// TIA Portal V20 export
FUNCTION_BLOCK "FB_Parameters"   // FB64, SCL
{ S7_Optimized_Access := 'TRUE' }
// stored: MemoryReserve 100, SetENOAutomatically false
   VAR
      Shuttle1Enable : "UDT_BoolEnable";
      Shuttle2Enable : Bool;
   END_VAR
   VAR RETAIN
      GazPressureManual : Real := 0.7;   // @Precision:3 @Unit:bar @Min:0.5 @Max:1.2
   END_VAR
   VAR
      CoolingVentilatorSetpoint : Real;
      TemperatureCoolingSetpoint : Real;
      BlowingSetpoint : Real;
      sPresenceShuttle1UndrilledPart : "FB_HMI_PLC_Pos";
      sPresenceShuttle1UndrilledBw { S7_SetPoint := 'True'} : "FB_HMI_PLC_Pos";
      sPresenceShuttle1DrilledPart { S7_SetPoint := 'True'} : "FB_HMI_PLC_Pos";
      sPresenceShuttle1DrilledBw { S7_SetPoint := 'True'} : "FB_HMI_PLC_Pos";
      sPresenceShuttle2UndrilledPart : "FB_HMI_PLC_Pos";
      sPresenceShuttle2UndrilledBw { S7_SetPoint := 'True'} : "FB_HMI_PLC_Pos";
      sPresenceShuttle2DrilledPart { S7_SetPoint := 'True'} : "FB_HMI_PLC_Pos";
      sPresenceShuttle2DrilledBw { S7_SetPoint := 'True'} : "FB_HMI_PLC_Pos";
      sPresenceGripperUndrilledPart : "FB_HMI_PLC_Pos";
      sPresenceGripperUndrilledBw { S7_SetPoint := 'True'} : "FB_HMI_PLC_Pos";
      sPresenceGripperDrilledPart { S7_SetPoint := 'True'} : "FB_HMI_PLC_Pos";
      sPresenceGripperDrilledBw { S7_SetPoint := 'True'} : "FB_HMI_PLC_Pos";
      sPresenceFixtureUndrilledPart : "FB_HMI_PLC_Pos";
      sPresenceFixtureUndrilledBw { S7_SetPoint := 'True'} : "FB_HMI_PLC_Pos";
      sPresenceFixtureDrilledPart { S7_SetPoint := 'True'} : "FB_HMI_PLC_Pos";
      sPresenceFixtureDrilledBw { S7_SetPoint := 'True'} : "FB_HMI_PLC_Pos";
      sHmiChangeEnable { S7_SetPoint := 'True'} : Bool;
   END_VAR
BEGIN
   REGION Description header 
       //==================================================================================
       // POSALUX Swiss SA / (C) Copyright 2025
       //----------------------------------------------------------------------------------
       // Title: FB_OPC_Parameters
       // Comment/Function: 
       // Author: Fabien WALDT
       // Engineering: TIA Portal v20
       //----------------------------------------------------------------------------------
       // Change log table:
       // Version  | Date     | Expert in charge | Changes applied
       // ---------|----------|------------------|-----------------------------------------
       // 00.00.01 | 20260304 | WFA              | First released version
       // =================================================================================
   END_REGION

   REGION Set Points (HMI -> PLC)
       "DB_HMISetting".GasAssistSetPoint := "DB_OPC_Machine".Parameters.GasAssistSetPoint;
       "DB_HMISetting".CoolingVentilatorSetpoint := "DB_OPC_Machine".Parameters.CoolingVentilatorSetpoint;
       "DB_HMISetting".TemperatureCoolingSetpoint := "DB_OPC_Machine".Parameters.TemperatureCoolingSetpoint;
       "DB_HMISetting".BlowingSetpoint := "DB_OPC_Machine".Parameters.BlowingSetpoint;
   END_REGION

   REGION Shuttle Enable (HMI -> PLC)
       "DB_OPC_Machine".Parameters.Shuttle1Enable.IsEnabled := NOT "DB_LoaderShuttle1".sMain.iJobReq AND NOT "DB_LoaderShuttle2".sMain.iJobReq;
       "DB_OPC_Machine".Parameters.Shuttle2Enable.IsEnabled := NOT "DB_LoaderShuttle1".sMain.iJobReq AND NOT "DB_LoaderShuttle2".sMain.iJobReq;

       "DB_HMISetting".Shuttle1Enable := "DB_OPC_Machine".Parameters.Shuttle1Enable.Value;
       "DB_HMISetting".Shuttle2Enable := "DB_OPC_Machine".Parameters.Shuttle2Enable.Value;
   END_REGION

   REGION Sequence
       // Shuttle 1
       "DB_OPC_Machine".Parameters.Sequence.Shuttle1.Main := "DB_LoaderShuttle1".sMain.sCurrent_Step_NB;
       "DB_OPC_Machine".Parameters.Sequence.Shuttle1.ShuttleInt := "DB_LoaderShuttle1".sShuttleInt.sCurrent_Step_NB;
       "DB_OPC_Machine".Parameters.Sequence.Shuttle1.ShuttleExt := "DB_LoaderShuttle1".sShuttleExt.sCurrent_Step_NB;
       "DB_OPC_Machine".Parameters.Sequence.Shuttle1.ControlIn := "DB_LoaderShuttle1".sControlIn.sCurrent_Step_NB;
       "DB_OPC_Machine".Parameters.Sequence.Shuttle1.ControlOut := "DB_LoaderShuttle1".sControlOut.sCurrent_Step_NB;
       "DB_OPC_Machine".Parameters.Sequence.Shuttle1.Blowing := "DB_LoaderShuttle1".sBlowing.sCurrent_Step_NB;
       "DB_OPC_Machine".Parameters.Sequence.Shuttle1.IntLoadUnload := "DB_LoaderShuttle1".sIntLoadUnload.sCurrent_Step_NB;
       "DB_OPC_Machine".Parameters.Sequence.Shuttle1.ExtLoadUnload := "DB_LoaderShuttle1".sExtLoadUnload.sCurrent_Step_NB;
       "DB_OPC_Machine".Parameters.Sequence.Shuttle1.BwLoadUnload := "DB_LoaderShuttle1".sBwLoadUnload.sCurrent_Step_NB;
       "DB_OPC_Machine".Parameters.Sequence.Shuttle1.BwControlIn := "DB_LoaderShuttle1".sBwControlIn.sCurrent_Step_NB;
       "DB_OPC_Machine".Parameters.Sequence.Shuttle1.ActControlIn := "DB_LoaderShuttle1".sActPartControlIn.sCurrent_Step_NB;
       "DB_OPC_Machine".Parameters.Sequence.Shuttle1.ActControlOut := "DB_LoaderShuttle1".sActPartControlOut.sCurrent_Step_NB;
       "DB_OPC_Machine".Parameters.Sequence.Shuttle1.ActBwControlIn := "DB_LoaderShuttle1".sActBwControlIn.sCurrent_Step_NB;

       // Shuttle 2
       "DB_OPC_Machine".Parameters.Sequence.Shuttle2.Main := "DB_LoaderShuttle2".sMain.sCurrent_Step_NB;
       "DB_OPC_Machine".Parameters.Sequence.Shuttle2.ShuttleInt := "DB_LoaderShuttle2".sShuttleInt.sCurrent_Step_NB;
       "DB_OPC_Machine".Parameters.Sequence.Shuttle2.ShuttleExt := "DB_LoaderShuttle2".sShuttleExt.sCurrent_Step_NB;
       "DB_OPC_Machine".Parameters.Sequence.Shuttle2.ControlIn := "DB_LoaderShuttle2".sControlIn.sCurrent_Step_NB;
       "DB_OPC_Machine".Parameters.Sequence.Shuttle2.ControlOut := "DB_LoaderShuttle2".sControlOut.sCurrent_Step_NB;
       "DB_OPC_Machine".Parameters.Sequence.Shuttle2.Blowing := "DB_LoaderShuttle2".sBlowing.sCurrent_Step_NB;
       "DB_OPC_Machine".Parameters.Sequence.Shuttle2.IntLoadUnload := "DB_LoaderShuttle2".sIntLoadUnload.sCurrent_Step_NB;
       "DB_OPC_Machine".Parameters.Sequence.Shuttle2.ExtLoadUnload := "DB_LoaderShuttle2".sExtLoadUnload.sCurrent_Step_NB;
       "DB_OPC_Machine".Parameters.Sequence.Shuttle2.BwLoadUnload := "DB_LoaderShuttle2".sBwLoadUnload.sCurrent_Step_NB;
       "DB_OPC_Machine".Parameters.Sequence.Shuttle2.BwControlIn := "DB_LoaderShuttle2".sBwControlIn.sCurrent_Step_NB;
       "DB_OPC_Machine".Parameters.Sequence.Shuttle2.ActControlIn := "DB_LoaderShuttle2".sActPartControlIn.sCurrent_Step_NB;
       "DB_OPC_Machine".Parameters.Sequence.Shuttle2.ActControlOut := "DB_LoaderShuttle2".sActPartControlout.sCurrent_Step_NB;
       "DB_OPC_Machine".Parameters.Sequence.Shuttle2.ActBwControlIn := "DB_LoaderShuttle2".sActBwControlIn.sCurrent_Step_NB;

       // Fixture
       "DB_OPC_Machine".Parameters.Sequence.Fixture.Blowing := "DB_LoaderFixture".sFixtureBlowing.sCurrent_Step_NB;
       "DB_OPC_Machine".Parameters.Sequence.Fixture.Loading := "DB_LoaderFixture".sFixtureLoading.sCurrent_Step_NB;
       "DB_OPC_Machine".Parameters.Sequence.Fixture.Unloading := "DB_LoaderFixture".sFixtureUnloading.sCurrent_Step_NB;
       "DB_OPC_Machine".Parameters.Sequence.Fixture.V_Init := "DB_LoaderFixture".sFixtureV_Init.sCurrent_Step_NB;
       "DB_OPC_Machine".Parameters.Sequence.Fixture.W_Init := "DB_LoaderFixture".sFixtureW_Init.sCurrent_Step_NB;

   END_REGION

   REGION Presence
       // Shuttle 1
        "DB_OPC_Machine".Parameters.Presence.Shuttle1UndrilledPart := "DB_PartManagement".sPosition.sShuttle1.Undrilled.Presence.Part;
        "DB_OPC_Machine".Parameters.Presence.Shuttle1UndrilledBw := "DB_PartManagement".sPosition.sShuttle1.Undrilled.Presence.BW;
        "DB_OPC_Machine".Parameters.Presence.Shuttle1DrilledPart := "DB_PartManagement".sPosition.sShuttle1.Drilled.Presence.Part;
        "DB_OPC_Machine".Parameters.Presence.Shuttle1DrilledBw := "DB_PartManagement".sPosition.sShuttle1.Drilled.Presence.BW;

       // Shuttle 2
       "DB_OPC_Machine".Parameters.Presence.Shuttle2UndrilledPart := "DB_PartManagement".sPosition.sShuttle2.Undrilled.Presence.Part;
       "DB_OPC_Machine".Parameters.Presence.Shuttle2UndrilledBw := "DB_PartManagement".sPosition.sShuttle2.Undrilled.Presence.BW;
       "DB_OPC_Machine".Parameters.Presence.Shuttle2DrilledPart := "DB_PartManagement".sPosition.sShuttle2.Drilled.Presence.Part;
       "DB_OPC_Machine".Parameters.Presence.Shuttle2DrilledBw := "DB_PartManagement".sPosition.sShuttle2.Drilled.Presence.BW;

       // Gripper
       "DB_OPC_Machine".Parameters.Presence.GripperUndrilledPart := "DB_PartManagement".sPosition.sGripper.Undrilled.Presence.Part;
       "DB_OPC_Machine".Parameters.Presence.GripperUndrilledBw := "DB_PartManagement".sPosition.sGripper.Undrilled.Presence.BW;
       "DB_OPC_Machine".Parameters.Presence.GripperDrilledPart := "DB_PartManagement".sPosition.sGripper.Drilled.Presence.Part;
       "DB_OPC_Machine".Parameters.Presence.GripperDrilledBw := "DB_PartManagement".sPosition.sGripper.Drilled.Presence.BW;

       // Fixture
       "DB_OPC_Machine".Parameters.Presence.FixtureUndrilledPart := "DB_PartManagement".sPosition.sFixture.Undrilled.Presence.Part;
       "DB_OPC_Machine".Parameters.Presence.FixtureUndrilledBw := "DB_PartManagement".sPosition.sFixture.Undrilled.Presence.BW;
       "DB_OPC_Machine".Parameters.Presence.FixtureDrilledPart := "DB_PartManagement".sPosition.sFixture.Drilled.Presence.Part;
       "DB_OPC_Machine".Parameters.Presence.FixtureDrilledBw := "DB_PartManagement".sPosition.sFixture.Drilled.Presence.BW;
   END_REGION

   REGION Presence V2
       // // Shuttle 1
       // #sPresenceShuttle1UndrilledPart("HMI_Change Enable" := #sHmiChangeEnable,
       //                                 ioPLC_State := "DB_PartManagement".sPosition.sShuttle1.Undrilled.Presence.Part,
       //                                 ioHMI_State := "DB_OPC_Machine".Parameters.Presence.Shuttle1UndrilledPart);

       // #sPresenceShuttle1UndrilledBw("HMI_Change Enable" := #sHmiChangeEnable,
       //                               ioPLC_State := "DB_PartManagement".sPosition.sShuttle1.Undrilled.Presence.BW,
       //                               ioHMI_State := "DB_OPC_Machine".Parameters.Presence.Shuttle1UndrilledBw);

       // #sPresenceShuttle1DrilledPart("HMI_Change Enable" := #sHmiChangeEnable,
       //                                 ioPLC_State := "DB_PartManagement".sPosition.sShuttle1.Drilled.Presence.Part,
       //                                 ioHMI_State := "DB_OPC_Machine".Parameters.Presence.Shuttle1DrilledPart);

       // #sPresenceShuttle1DrilledBw("HMI_Change Enable" := #sHmiChangeEnable,
       //                               ioPLC_State := "DB_PartManagement".sPosition.sShuttle1.Drilled.Presence.BW,
       //                               ioHMI_State := "DB_OPC_Machine".Parameters.Presence.Shuttle1DrilledBw);

       //  // Shuttle 2
       //  #sPresenceShuttle2UndrilledPart("HMI_Change Enable" := #sHmiChangeEnable,
       //                                  ioPLC_State := "DB_PartManagement".sPosition.sShuttle2.Undrilled.Presence.Part,
       //                                  ioHMI_State := "DB_OPC_Machine".Parameters.Presence.Shuttle2UndrilledPart);

       //  #sPresenceShuttle2UndrilledBw("HMI_Change Enable" := #sHmiChangeEnable,
       //                                ioPLC_State := "DB_PartManagement".sPosition.sShuttle2.Undrilled.Presence.BW,
       //                                ioHMI_State := "DB_OPC_Machine".Parameters.Presence.Shuttle2UndrilledBw);

       //  #sPresenceShuttle2DrilledPart("HMI_Change Enable" := #sHmiChangeEnable,
       //                                ioPLC_State := "DB_PartManagement".sPosition.sShuttle2.Drilled.Presence.Part,
       //                                ioHMI_State := "DB_OPC_Machine".Parameters.Presence.Shuttle2DrilledPart);

       //  #sPresenceShuttle2DrilledBw("HMI_Change Enable" := #sHmiChangeEnable,
       //                              ioPLC_State := "DB_PartManagement".sPosition.sShuttle2.Drilled.Presence.BW,
       //                              ioHMI_State := "DB_OPC_Machine".Parameters.Presence.Shuttle2DrilledBw);

       //  // Gripper
       //  #sPresenceGripperUndrilledPart("HMI_Change Enable" := #sHmiChangeEnable,
       //                                 ioPLC_State := "DB_PartManagement".sPosition.sGripper.Undrilled.Presence.Part,
       //                                 ioHMI_State := "DB_OPC_Machine".Parameters.Presence.GripperUndrilledPart);

       //  #sPresenceGripperUndrilledBw("HMI_Change Enable" := #sHmiChangeEnable,
       //                               ioPLC_State := "DB_PartManagement".sPosition.sGripper.Undrilled.Presence.BW,
       //                               ioHMI_State := "DB_OPC_Machine".Parameters.Presence.GripperUndrilledBw);

       //  #sPresenceGripperDrilledPart("HMI_Change Enable" := #sHmiChangeEnable,
       //                               ioPLC_State := "DB_PartManagement".sPosition.sGripper.Drilled.Presence.Part,
       //                               ioHMI_State := "DB_OPC_Machine".Parameters.Presence.GripperDrilledPart);

       //  #sPresenceGripperDrilledBw("HMI_Change Enable" := #sHmiChangeEnable,
       //                             ioPLC_State := "DB_PartManagement".sPosition.sGripper.Drilled.Presence.BW,
       //                             ioHMI_State := "DB_OPC_Machine".Parameters.Presence.GripperDrilledBw);

       //  // Fixture
       //  #sPresenceFixtureUndrilledPart("HMI_Change Enable" := #sHmiChangeEnable,
       //                                 ioPLC_State := "DB_PartManagement".sPosition.sFixture.Undrilled.Presence.Part,
       //                                 ioHMI_State := "DB_OPC_Machine".Parameters.Presence.FixtureUndrilledPart);

       //  #sPresenceFixtureUndrilledBw("HMI_Change Enable" := #sHmiChangeEnable,
       //                               ioPLC_State := "DB_PartManagement".sPosition.sFixture.Undrilled.Presence.BW,
       //                               ioHMI_State := "DB_OPC_Machine".Parameters.Presence.FixtureUndrilledBw);

       //  #sPresenceFixtureDrilledPart("HMI_Change Enable" := #sHmiChangeEnable,
       //                               ioPLC_State := "DB_PartManagement".sPosition.sFixture.Drilled.Presence.Part,
       //                               ioHMI_State := "DB_OPC_Machine".Parameters.Presence.FixtureDrilledPart);

       //  #sPresenceFixtureDrilledBw("HMI_Change Enable" := #sHmiChangeEnable,
       //                             ioPLC_State := "DB_PartManagement".sPosition.sFixture.Drilled.Presence.BW,
       //                             ioHMI_State := "DB_OPC_Machine".Parameters.Presence.FixtureDrilledBw);
   END_REGION
END_FUNCTION_BLOCK
